TYPE AlarmParameters :
STRUCT
	Control: AlarmControl;
	Enabled: AlarmSignals := ( 	A := ( 		
										FireExtract := TRUE,
										FireExtractTemperature := TRUE,
										FireExtractPressure := TRUE,
										FireExtractExternal := TRUE,
										FireLocal := TRUE,
										FireSupply := TRUE,
										Freeze := TRUE,
										Fuse := TRUE,
										Cold := TRUE,
										Aux := TRUE
									),
									B := (	
										RegulationDeviation := TRUE,
										SupplyAirDeviation := TRUE,
										ExtractAirDeviation := TRUE,
										SupplyFan := TRUE,
										ExtractFan := TRUE,
										HeatExchangerEfficiency := TRUE,
										Defrost := TRUE,
										SupplyFilter := TRUE,
										ExtractFilter := TRUE,
										SmokeDetectorServiceSupply := TRUE,
										SmokeDetectorServiceExtract := TRUE,
										Pump1 := TRUE,
										DamperError := TRUE,
										CommunicationError := TRUE,
										DamperModuleService := TRUE
									),
									C := (	
										ExternalSmokeControl := TRUE,
										ModbusRTU := TRUE,
										ModbusTCP := TRUE,
										SensorFailure := TRUE
									));
	AutoReset: AlarmSignals := ( 	A := ( 	FirePanelSupplyStart := TRUE,  
											FirePanelSupplyStop := TRUE, 
											FirePanelExtractStart := TRUE, 
											FirePanelExtractStop := TRUE,
											Fuse := TRUE,
											AL01 := TRUE,
											AL02 := TRUE,
											AL03 := TRUE,
											AL04 := TRUE,
											AL05 := TRUE,
											AL06 := TRUE,
											AL07 := TRUE,
											AL08 := TRUE
									),
									B := (	RegulationDeviation := TRUE,
											SupplyAirDeviation := TRUE,
											ExtractAirDeviation := TRUE,
											SupplyFan := FALSE,
											ExtractFan := FALSE,
											HeatExchangerEfficiency := TRUE,
											Defrost := TRUE,
											SupplyFilter := TRUE,
											ExtractFilter := TRUE,
											SmokeDetectorServiceSupply := TRUE,
											Pump1 := TRUE,
											Pump2 := TRUE,
											CommunicationError := TRUE
									),
									C := (	ExternalSmokeControl := TRUE,
											ModbusRTU := TRUE,
											ModbusTCP := TRUE,
											SensorFailure := TRUE
									));
	Limits: AlarmLimits;
	Delay: AlarmDelays; // MUST be in same order and number as AlarmSignals
	Polarity: AlarmSignals := ( A:= ( FireExtract := FALSE ));
	Active: AlarmSignals;
	Status: AlarmSignals;	
	
END_STRUCT
END_TYPE

(* stored: Version 1.1.0.1, ProductVersion 3.1.4024.6
   DUT AlarmParameters: Id {b930426d-7843-4419-9378-33c5b23e1312} *)
